(* Logix 5000 project; controller Safety vendor 1 type 14 code 148 rev 32.11; software revision 32.03; part 16 of 17 *)
(* tags used below, declared in another part *)
   A1_CoilCarSolPwrEn : BOOL;   // A1 UNW COIL CAR Solenoid Safe-Off Enable ( 1= Enable )
   A1_S20_ModFlt : ALIAS FOR Flt_Modules[0].0;   // A1 Point I/O Slot20 Module Fault (1 = Fault)
   A1_S21_ModFlt : ALIAS FOR Flt_Modules[0].1;   // A1 Point I/O Slot21 Module Fault (1 = Fault)
   C1_S12_ModFlt : ALIAS FOR Flt_Modules[0].2;   // C1 Point I/O Slot12 Module Fault (1 = Fault)
   CC : ALIAS FOR Diag_Tmp.0;   // Chris Como's Test Bit Always On Bit
   CHPLC_S1_ModFlt : ALIAS FOR Flt_Modules[0].3;   // CHPLC Point I/O Slot01 Module Fault (1 = Fault)
   CHPLC_S2_ModFlt : ALIAS FOR Flt_Modules[0].4;   // CHPLC Point I/O Slot02 Module Fault (1 = Fault)
   CHPLC_S3_ModFlt : ALIAS FOR Flt_Modules[0].5;   // CHPLC Point I/O Slot03 Module Fault (1 = Fault)
   CHPLC_S4_ModFlt : ALIAS FOR Flt_Modules[0].6;   // CHPLC Point I/O Slot04 Module Fault (1 = Fault)
   CHPLC_S5_ModFlt : ALIAS FOR Flt_Modules[0].7;   // CHPLC Point I/O Slot05 Module Fault (1 = Fault)
   CHPLC_S6_ModFlt : ALIAS FOR Flt_Modules[0].8;   // CHPLC Point I/O Slot06 Module Fault (1 = Fault)
   Citect_HB_Flt : BOOL;   // Citect Heartbeat Fault ( 1= Fault)
   Citect_HB_TOF : TIMER;   // Citect Heartbeat Timer Off
   Citect_HB_TON : TIMER;   // Citect Heartbeat Timer On
   D1_S12_ModFlt : ALIAS FOR Flt_Modules[0].9;   // D1 Point I/O Slot12 Module Fault (1 = Fault)
   DPD_No_EStops : BOOL;   // DPD No Estops ( 1= OK)
   DPD_S14_ModFlt : ALIAS FOR Flt_Modules[0].10;   // DPD Point I/O Slot14 Module Fault (1 = Fault)
   DPD_S15_ModFlt : ALIAS FOR Flt_Modules[0].11;   // DPD Point I/O Slot15 Module Fault (1 = Fault)
   Drives_Off : DINT;   // Line Drives Off
   E1_S10_ModFlt : ALIAS FOR Flt_Modules[0].12;   // E1 Point I/O Slot10 Module Fault (1 = Fault)
   EnBridle_DrvsOff : BOOL;   // Entry Bridle Drives OFF ( 1= OFF)
   ESTOP_x201PB040_Flt : ALIAS FOR Flt_Estops.0;   // OS1 Line EStop Pushbutton Fault ( 1= Fault)
   ESTOP_x211PB040_Flt : ALIAS FOR Flt_Estops.1;   // OS2 Line EStop Pushbutton Fault ( 1= Fault)
   ESTOP_x221PB040_Flt : ALIAS FOR Flt_Estops.2;   // OS3 Line EStop Pushbutton Fault ( 1= Fault)
   ESTOP_x231PB040_Flt : ALIAS FOR Flt_Estops.3;   // OS4N Line EStop Pushbutton Fault ( 1= Fault)
   ESTOP_x241PB040_Flt : ALIAS FOR Flt_Estops.4;   // OS4S Line EStop Pushbutton Fault ( 1= Fault)
   ESTOP_x251PB040_Flt : ALIAS FOR Flt_Estops.5;   // OS5 Line EStop Pushbutton Fault ( 1= Fault)
   ESTOP_x261PB040_Flt : ALIAS FOR Flt_Estops.6;   // OS6 Line EStop Pushbutton Fault ( 1= Fault)
   ESTOP_x271PB040_Flt : ALIAS FOR Flt_Estops.7;   // OS8 Line EStop Pushbutton Fault ( 1= Fault)
   ESTOP_x281PB040_Flt : ALIAS FOR Flt_Estops.8;   // OS9 Line EStop Pushbutton Fault ( 1= Fault)
   ESTOP_x291PB040_Flt : ALIAS FOR Flt_Estops.9;   // OS11 Line EStop Pushbutton Fault ( 1= Fault)
   ESTOP_x301PB040_Flt : ALIAS FOR Flt_Estops.10;   // OS13 Line EStop Pushbutton Fault ( 1= Fault)
   ESTOP_x311PB040_Flt : ALIAS FOR Flt_Estops.11;   // OS14 Line EStop Pushbutton Fault ( 1= Fault)
   ESTOP_x311PB130_Flt : ALIAS FOR Flt_Estops.17;   // OS14 Shear EStop Pushbutton Fault ( 1= Fault)
   ESTOP_x321PB040_Flt : ALIAS FOR Flt_Estops.12;   // OS15 Line EStop Pushbutton Fault ( 1= Fault)
   ESTOP_x331PB040_Flt : ALIAS FOR Flt_Estops.13;   // OS16 Line EStop Pushbutton Fault ( 1= Fault)
   ESTOP_x480PB470_Flt : ALIAS FOR Flt_Estops.14;   // DPD Line EStop Pushbutton Fault ( 1= Fault)
   ESTOP_x519LS470_Flt : ALIAS FOR Flt_Estops.18;   // G1 Line EStop Tripwire Limit Switch Fault ( 1= Fault)
   ESTOP_x533PB470_Flt : ALIAS FOR Flt_Estops.16;   // H1 Line EStop Pushbutton Fault ( 1= Fault)
   ExBridle_DrvsOff : BOOL;   // Exit Bridle Drives OFF ( 1= OFF)
   F1_S19_ModFlt : ALIAS FOR Flt_Modules[0].13;   // F1 Point I/O Slot19 Module Fault (1 = Fault)
   F1_S20_ModFlt : ALIAS FOR Flt_Modules[0].14;   // F1 Point I/O Slot20 Module Fault (1 = Fault)
   FromMachine : DINT[35];   // (FromMach)
   FromSafety : DINT[35];   // (From Safety)
   FromShearDie : DINT[35];   // (From Shear Die)
   FVR_y702MTR191_Flt : ALIAS FOR Flt_Starter.4;   // Rewind Pinch Roll Starter Fault ( 1= Fault)
   FVR_y708MTR080_Flt : ALIAS FOR Flt_Starter.1;   // Flattener Drive Motor Starter Fault ( 1= Fault)
   FVR_y708MTR250_Flt : ALIAS FOR Flt_Starter.0;   // Unwind Hold Down Roll Starter Fault ( 1= Fault)
   FVR_y753MTR190_Flt : ALIAS FOR Flt_Starter.2;   // Trimmer Pinch Roll Starter Fault ( 1= Fault)
   FVR_y761MTR081_Flt : ALIAS FOR Flt_Starter.3;   // Trimmer Scrap Conveyor Starter Fault ( 1= Fault)
   FVR_y778MTR080_Flt : ALIAS FOR Flt_Starter.5;   // Shear Die Crank Starter Fault ( 1= Fault)
   FVR_y802MTR080_Flt : ALIAS FOR Flt_Starter.6;   // Stacker Side Guide Lift Starter Fault ( 1= Fault)
   FVR_y802MTR230_Flt : ALIAS FOR Flt_Starter.8;   // Scrap Horizontal Conveyor Starter Fault ( 1= Fault)
   FVR_y802MTR231_Flt : ALIAS FOR Flt_Starter.7;   // Stacker Chain Conveyor Starter Fault ( 1= Fault)
   G1_No_EStops : BOOL;   // G1 No Estops ( 1= OK)
   G1_S11_ModFlt : ALIAS FOR Flt_Modules[0].15;   // G1 Point I/O Slot11 Module Fault (1 = Fault)
   G1_S12_ModFlt : ALIAS FOR Flt_Modules[0].16;   // G1 Point I/O Slot12 Module Fault (1 = Fault)
   H1_No_EStops : BOOL;   // H1 No Estops ( 1= OK)
   H1_S5_ModFlt : ALIAS FOR Flt_Modules[0].17;   // H1 Point I/O Slot05 Module Fault (1 = Fault)
   H1_S6_ModFlt : ALIAS FOR Flt_Modules[0].18;   // H1 Point I/O Slot06 Module Fault (1 = Fault)
   HB_Citect : BOOL;   // Heartbeat Citect Reflect
   Line_CTC_CoastStop : BOOL;   // Line Coast Stop ( 1= Coast Stop) (Condition Exists)
   Line_CTL_CoastStop : BOOL;   // Line Coast Stop ( 1= Coast Stop) (Condition Exists)
   Line_NoP2P_CommFlts : BOOL;   // Line No Peer to Peer Comm Faults ( 1= OK)
   Line_Total_CoastStop : BOOL;   // Line Coast Stop ( 1= Coast Stop) (Condition Exists)
   Line_TotalMode : BOOL;   // Line TOTAL Mode ( 1= Total Mode) (0 = Coil to Coil)
   LineSts : UDT_SysStatus;
   Machine_HB_Flt : BOOL;   // Machine Heartbeat Fault ( 1= Fault)
   Machine_HB_TOF : TIMER;   // Machine Heartbeat Timer Off
   Machine_HB_TON : TIMER;   // Machine Heartbeat Timer On
   MCC1_S1_ModFlt : ALIAS FOR Flt_Modules[2].0;   // MCC1 Point I/O Slot01 Module Fault (1 = Fault)
   MCC1_S6_ModFlt : ALIAS FOR Flt_Modules[2].1;   // MCC1 Point I/O Slot06 Module Fault (1 = Fault)
   MCC2_S1_ModFlt : ALIAS FOR Flt_Modules[2].2;   // MCC2 Point I/O Slot01 Module Fault (1 = Fault)
   MCC2_S2_ModFlt : ALIAS FOR Flt_Modules[2].3;   // MCC2 Point I/O Slot02 Module Fault (1 = Fault)
   MCC3_S1_ModFlt : ALIAS FOR Flt_Modules[2].4;   // MCC3 Point I/O Slot01 Module Fault (1 = Fault)
   MCC3_S3_ModFlt : ALIAS FOR Flt_Modules[2].5;   // MCC3 Point I/O Slot03 Module Fault (1 = Fault)
   MCC3_S4_ModFlt : ALIAS FOR Flt_Modules[2].6;   // MCC3 Point I/O Slot04 Module Fault (1 = Fault)
   MCC4_S1_ModFlt : ALIAS FOR Flt_Modules[2].7;   // MCC4 Point I/O Slot01 Module Fault (1 = Fault)
   MCC4_S3_ModFlt : ALIAS FOR Flt_Modules[2].8;   // MCC4 Point I/O Slot03 Module Fault (1 = Fault)
   MCC4_S4_ModFlt : ALIAS FOR Flt_Modules[2].9;   // MCC4 Point I/O Slot04 Module Fault (1 = Fault)
   MCC5_S1_ModFlt : ALIAS FOR Flt_Modules[2].10;   // MCC5 Point I/O Slot01 Module Fault (1 = Fault)
   MCC5_S3_ModFlt : ALIAS FOR Flt_Modules[2].11;   // MCC5 Point I/O Slot03 Module Fault (1 = Fault)
   MCC5_S4_ModFlt : ALIAS FOR Flt_Modules[2].12;   // MCC5 Point I/O Slot04 Module Fault (1 = Fault)
   MCC5_S5_ModFlt : ALIAS FOR Flt_Modules[2].13;   // MCC5 Point I/O Slot05 Module Fault (1 = Fault)
   OS11_No_EStops : BOOL;   // OS11 No Estops ( 1= OK)
   OS11_S1_ModFlt : ALIAS FOR Flt_Modules[1].11;   // OS11 Point I/O Slot01 Module Fault (1 = Fault)
   OS13_No_EStops : BOOL;   // OS13 No Estops ( 1= OK)
   OS13_S1_ModFlt : ALIAS FOR Flt_Modules[1].12;   // OS13 Point I/O Slot01 Module Fault (1 = Fault)
   OS14_No_EStops : BOOL;   // OS14 No Estops ( 1= OK)
   OS14_S1_ModFlt : ALIAS FOR Flt_Modules[1].13;   // OS14 Point I/O Slot01 Module Fault (1 = Fault)
   OS14_Shear_No_EStops : BOOL;   // OS14_Shear No Estops ( 1= OK)
   OS15_No_EStops : BOOL;   // OS15 No Estops ( 1= OK)
   OS15_S1_ModFlt : ALIAS FOR Flt_Modules[1].14;   // OS15 Point I/O Slot01 Module Fault (1 = Fault)
   OS16_No_EStops : BOOL;   // OS16 No Estops ( 1= OK)
   OS16_S1_ModFlt : ALIAS FOR Flt_Modules[1].15;   // OS16 Point I/O Slot01 Module Fault (1 = Fault)
   OS1_No_EStops : BOOL;   // OS1 No Estops ( 1= OK)
   OS1_S1_ModFlt : ALIAS FOR Flt_Modules[1].0;   // OS1 Point I/O Slot01 Module Fault (1 = Fault)
   OS2_No_EStops : BOOL;   // OS2 No Estops ( 1= OK)
   OS2_S1_ModFlt : ALIAS FOR Flt_Modules[1].1;   // OS2 Point I/O Slot01 Module Fault (1 = Fault)
   OS3_No_EStops : BOOL;   // OS3 No Estops ( 1= OK)
   OS3_S1_ModFlt : ALIAS FOR Flt_Modules[1].2;   // OS3 Point I/O Slot01 Module Fault (1 = Fault)
   OS4_No_EStops : BOOL;   // OS4 No Estops ( 1= OK)
   OS4N_S1_ModFlt : ALIAS FOR Flt_Modules[1].3;   // OS4N Point I/O Slot01 Module Fault (1 = Fault)
   OS4N_S5_ModFlt : ALIAS FOR Flt_Modules[1].4;   // OS4N Point I/O Slot05 Module Fault (1 = Fault)
   OS4S_S1_ModFlt : ALIAS FOR Flt_Modules[1].5;   // OS4S Point I/O Slot01 Module Fault (1 = Fault)
   OS4S_S5_ModFlt : ALIAS FOR Flt_Modules[1].6;   // OS4S Point I/O Slot05 Module Fault (1 = Fault)
   OS5_No_EStops : BOOL;   // OS5 No Estops ( 1= OK)
   OS5_S1_ModFlt : ALIAS FOR Flt_Modules[1].7;   // OS5 Point I/O Slot01 Module Fault (1 = Fault)
   OS6_No_EStops : BOOL;   // OS6 No Estops ( 1= OK)
   OS6_S1_ModFlt : ALIAS FOR Flt_Modules[1].8;   // OS6 Point I/O Slot01 Module Fault (1 = Fault)
   OS8_No_EStops : BOOL;   // OS8 No Estops ( 1= OK)
   OS8_S1_ModFlt : ALIAS FOR Flt_Modules[1].9;   // OS8 Point I/O Slot01 Module Fault (1 = Fault)
   OS9_No_EStops : BOOL;   // OS9 No Estops ( 1= OK)
   OS9_S1_ModFlt : ALIAS FOR Flt_Modules[1].10;   // OS9 Point I/O Slot01 Module Fault (1 = Fault)
   PrCon_DrvsOff : BOOL;   // Product Conveyors (1-3) Drives OFF ( 1= OFF)
   PW_DrvsOff : BOOL;   // Paper Winder Drives OFF ( 1= OFF)
   Rew_DrvsOff : BOOL;   // Rewind Drives OFF ( 1= OFF)
   SafeOff_y172CR460_Flt : ALIAS FOR Flt_SafeOff[0].0;   // Shear Die Main Contactor Relay Fault ( 1= Fault)
   SafeOff_y172CR510_Flt : ALIAS FOR Flt_SafeOff[0].1;   // Shear Die Drive Enable Relay Fault ( 1= Fault)
   SafeOff_y613CR460_Flt : ALIAS FOR Flt_SafeOff[0].2;   // Unwind Op Side Main Contactor Relay Fault ( 1= Fault)
   SafeOff_y613CR510_Flt : ALIAS FOR Flt_SafeOff[0].3;   // Unwind Op Side Drive Enable Relay Fault ( 1= Fault)
   SafeOff_y613CR550_Flt : ALIAS FOR Flt_SafeOff[0].4;   // Unwind Drive Side Main Contactor Relay Fault ( 1= Fault)
   SafeOff_y613CR590_Flt : ALIAS FOR Flt_SafeOff[0].5;   // Unwind Drive Side Drive Enable Relay Fault ( 1= Fault)
   SafeOff_y613CR630_Flt : ALIAS FOR Flt_SafeOff[0].6;   // #1 Entry Bridle Roll 2 Main Contactor Relay Fault ( 1= Fault)
   SafeOff_y613CR670_Flt : ALIAS FOR Flt_SafeOff[0].7;   // #1 Entry Bridle Roll 2 Drive Enable Relay Fault ( 1= Fault)
   SafeOff_y613CR710_Flt : ALIAS FOR Flt_SafeOff[0].8;   // #2 Entry Bridle Roll 3 Main Contactor Relay Fault ( 1= Fault)
   SafeOff_y613CR750_Flt : ALIAS FOR Flt_SafeOff[0].9;   // #2 Entry Bridle Roll 3 Drive Enable Relay Fault ( 1= Fault)
   SafeOff_y614CR040_Flt : ALIAS FOR Flt_SafeOff[0].10;   // #1 Exit Bridle Roll 6 Main Contactor Relay Fault ( 1= Fault)
   SafeOff_y614CR090_Flt : ALIAS FOR Flt_SafeOff[0].11;   // #1 Exit Bridle Roll 6 Drive Enable Relay Fault ( 1= Fault)
   SafeOff_y614CR130_Flt : ALIAS FOR Flt_SafeOff[0].12;   // #2 Exit Bridle Roll 7 Main Contactor Relay Fault ( 1= Fault)
   SafeOff_y614CR170_Flt : ALIAS FOR Flt_SafeOff[0].13;   // #2 Exit Bridle Roll 7 Drive Enable Relay Fault ( 1= Fault)
   SafeOff_y614CR210_Flt : ALIAS FOR Flt_SafeOff[0].14;   // Rewind Main Contactor Relay Fault ( 1= Fault)
   SafeOff_y614CR250_Flt : ALIAS FOR Flt_SafeOff[0].15;   // Rewind Drive Enable Relay Fault ( 1= Fault)
   Safety_HB_TOF : TIMER;   // Safety Heartbeat Pulse Time Off
   Safety_HB_TON : TIMER;   // Safety Heartbeat Pulse Time On
   SC_DrvsOff : BOOL;   // Scrap Chop Conveyor Drives OFF ( 1= OFF)
   ScInCon_DrvsOff : BOOL;   // Scrap Incline Conveyor Drives OFF ( 1= OFF)
   SDPLC_S1_ModFlt : ALIAS FOR Flt_Modules[0].19;   // SDPLC Point I/O Slot01 Module Fault (1 = Fault)
   SDPLC_S2_ModFlt : ALIAS FOR Flt_Modules[0].20;   // SDPLC Point I/O Slot02 Module Fault (1 = Fault)
   Sfty_InstrFlts0_CTC : BOOL;   // Coil To Coil Estop Safety Instructions OK ( 1= No Faults)
   Sfty_InstrFlts0_CTL : BOOL;   // Cut To Length Estop Safety Instructions OK ( 1= No Faults)
   Sfty_InstrFlts0_Total : BOOL;   // Total Mode Estop Safety Instructions OK ( 1= No Faults)
   Sfty_InstrFlts1_CTC : BOOL;   // Coil To Coil Safe-Off Safety Instructions OK ( 1= No Faults)
   Sfty_InstrFlts1_CTL : BOOL;   // Cut To Length Safe-Off Safety Instructions OK ( 1= No Faults)
   Sfty_InstrFlts1_Total : BOOL;   // Total Mode Safe-Off Safety Instructions OK ( 1= No Faults)
   Sfty_InstrFlts2_CTC : BOOL;   // Coil To Coil FVR/FVNR Starters Safety Instructions OK ( 1= No Faults)
   Sfty_InstrFlts2_CTL : BOOL;   // Cut To Length FVR/FVNR Starters Safety Instructions OK ( 1= No Faults)
   Sfty_InstrFlts2_Total : BOOL;   // Total Mode FVR/FVNR Starters Safety Instructions OK ( 1= No Faults)
   Sfty_ModFlts0_CTC : BOOL;   // Coil To Coil General I/O Safety Module Faults ( 1= OK)
   Sfty_ModFlts0_CTL : BOOL;   // Cut To Length General I/O Safety Module Faults ( 1= OK)
   Sfty_ModFlts0_Total : BOOL;   // Total Mode General I/O Safety Module Faults ( 1= OK)
   Sfty_ModFlts1_CTC : BOOL;   // Coil To Coil Operator Station Safety Module Faults ( 1= OK)
   Sfty_ModFlts1_CTL : BOOL;   // Cut To Length Operator Station Safety Module Faults ( 1= OK)
   Sfty_ModFlts1_Total : BOOL;   // Total Mode Operator Station Safety Module Faults ( 1= OK)
   Sfty_ModFlts2_CTC : BOOL;   // Coil To Coil MCC Safety Module Faults ( 1= OK)
   Sfty_ModFlts2_CTL : BOOL;   // Cut To Lenght MCC Safety Module Faults ( 1= OK)
   Sfty_ModFlts2_Total : BOOL;   // Total Mode MCC Safety Module Faults ( 1= OK)
   SftyMap_Citect : DINT[5];   // SAFETY MAPPED From Citect System
   SftyMap_Mach : DINT[5];   // SAFETY MAPPED From Machine Processor
   SftyMap_ShDie : DINT[5];   // SAFETY MAPPED From Shear Die Processor
   SGWA_DrvsOff : BOOL;   // Side Guide Width Adjust Drives OFF ( 1= OFF)
   Shear_CoastStop : BOOL;   // Shear Coast Stop ( 1= Coast Stop) (Condition Exists)
   Shear_HB_Flt : BOOL;   // Shear Heartbeat Fault ( 1= Fault)
   Shear_HB_TOF : TIMER;   // Shear Heartbeat Pulse Time Off
   Shear_HB_TON : TIMER;   // Shear Heartbeat Pulse Time On
   ShearSts : UDT_ShearStatus;
   SkBkSt_DrvsOff : BOOL;   // Stacker Backstop Drives OFF ( 1= OFF)
   SkBlwr_DrvsOff : BOOL;   // Stacker Blower Drives OFF ( 1= OFF)
   Sr_DrvsOff : BOOL;   // Shear Pinch Roll/ Metering Back Up Drives OFF ( 1= OFF)
   SrCon_DrvsOff : BOOL;   // Shear Conveyor Drives OFF ( 1= OFF)
   SrDie_DrvsOff : BOOL;   // Shear Die Drives OFF ( 1= OFF)
   StPR_DrvsOff : BOOL;   // Sheeter Pinch Roll Drives OFF ( 1= OFF)
   TK_DrvsOff : BOOL;   // Trimmer Knives/ Width Adjust Drives OFF ( 1= OFF)
   ToCitect : DINT[64];   // (To Citect)
   UnPR_DrvsOff : BOOL;   // Unwind Pinch Roll Drives OFF ( 1= OFF)
   UNW_DrvsOff : BOOL;   // Unwind Drives OFF ( 1= OFF)
   VS2_S10_ModFlt : ALIAS FOR Flt_Modules[0].21;   // VS2 Point I/O Slot10 Module Fault (1 = Fault)
   WTPR_DrvsOff : BOOL;   // Wash Tank Pinch Rolls (1-4) Drives OFF ( 1= OFF)
(* System, continued *)

ROUTINE A04_SftyHeartbeat   (* ladder *)
// Heartbeat Logic
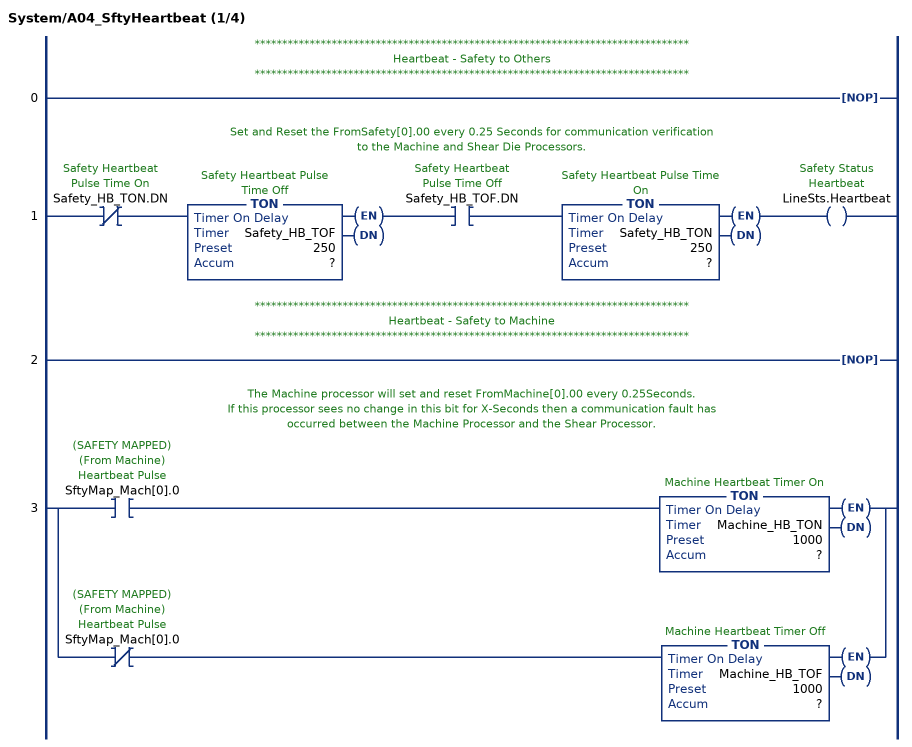
   // *******************************************************************************
   // Heartbeat - Safety to Others
   // *******************************************************************************
   0: NOP();
   // Set and Reset the FromSafety[0].00 every 0.25 Seconds for communication verification
   // to the Machine and Shear Die Processors.
   1: XIO(Safety_HB_TON.DN)TON(Safety_HB_TOF,?,?)XIC(Safety_HB_TOF.DN)TON(Safety_HB_TON,?,?)OTE(LineSts.Heartbeat);
   // *******************************************************************************
   // Heartbeat - Safety to Machine
   // *******************************************************************************
   2: NOP();
   // The Machine processor will set and reset FromMachine[0].00 every 0.25Seconds.
   // If this processor sees no change in this bit for X-Seconds then a communication fault has
   // occurred between the Machine Processor and the Shear Processor.
   3: [XIC(SftyMap_Mach[0].0) TON(Machine_HB_TON,?,?) ,XIO(SftyMap_Mach[0].0) TON(Machine_HB_TOF,?,?) ];
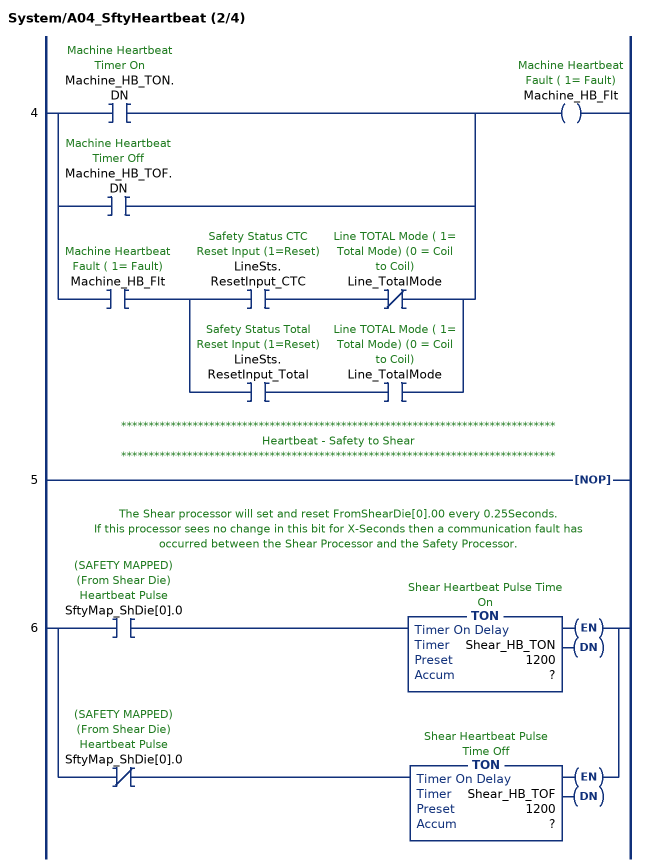
   4: [XIC(Machine_HB_TON.DN) ,XIC(Machine_HB_TOF.DN) ,XIC(Machine_HB_Flt) [XIC(LineSts.ResetInput_CTC) XIO(Line_TotalMode) ,XIC(LineSts.ResetInput_Total) XIC(Line_TotalMode) ] ]OTE(Machine_HB_Flt);
   // *******************************************************************************
   // Heartbeat - Safety to Shear
   // *******************************************************************************
   5: NOP();
   // The Shear processor will set and reset FromShearDie[0].00 every 0.25Seconds.
   // If this processor sees no change in this bit for X-Seconds then a communication fault has
   // occurred between the Shear Processor and the Safety Processor.
   6: [XIC(SftyMap_ShDie[0].0) TON(Shear_HB_TON,?,?) ,XIO(SftyMap_ShDie[0].0) TON(Shear_HB_TOF,?,?) ];
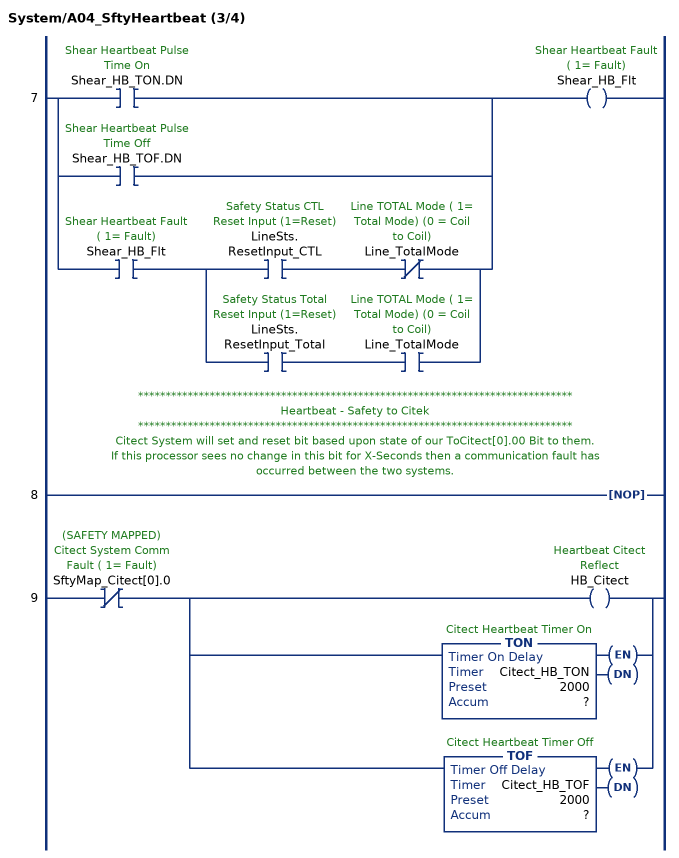
   7: [XIC(Shear_HB_TON.DN) ,XIC(Shear_HB_TOF.DN) ,XIC(Shear_HB_Flt) [XIC(LineSts.ResetInput_CTL) XIO(Line_TotalMode) ,XIC(LineSts.ResetInput_Total) XIC(Line_TotalMode) ] ]OTE(Shear_HB_Flt);
   // *******************************************************************************
   // Heartbeat - Safety to Citek
   // *******************************************************************************
   // Citect System will set and reset bit based upon state of our ToCitect[0].00 Bit to them.
   // If this processor sees no change in this bit for X-Seconds then a communication fault has
   // occurred between the two systems.
   8: NOP();
   9: XIO(SftyMap_Citect[0].0)[OTE(HB_Citect) ,TON(Citect_HB_TON,?,?) ,TOF(Citect_HB_TOF,?,?) ];
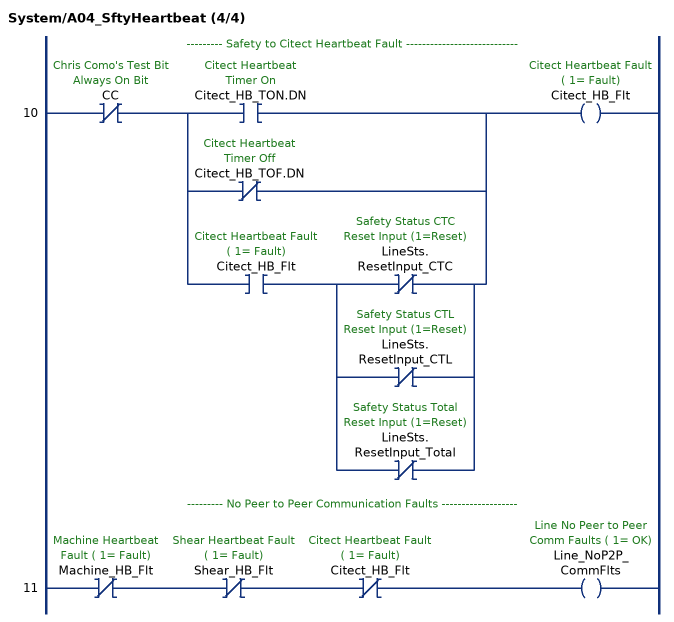
   // --------- Safety to Citect Heartbeat Fault ----------------------------
   10: XIO(CC)[XIC(Citect_HB_TON.DN) ,XIO(Citect_HB_TOF.DN) ,XIC(Citect_HB_Flt) [XIO(LineSts.ResetInput_CTC) ,XIO(LineSts.ResetInput_CTL) ,XIO(LineSts.ResetInput_Total) ] ]OTE(Citect_HB_Flt);
   // --------- No Peer to Peer Communication Faults -------------------
   11: XIO(Machine_HB_Flt)XIO(Shear_HB_Flt)XIO(Citect_HB_Flt)OTE(Line_NoP2P_CommFlts);
END_ROUTINE

ROUTINE B00_Line_Logic   (* ladder *)
// Line System
// Safety Logic
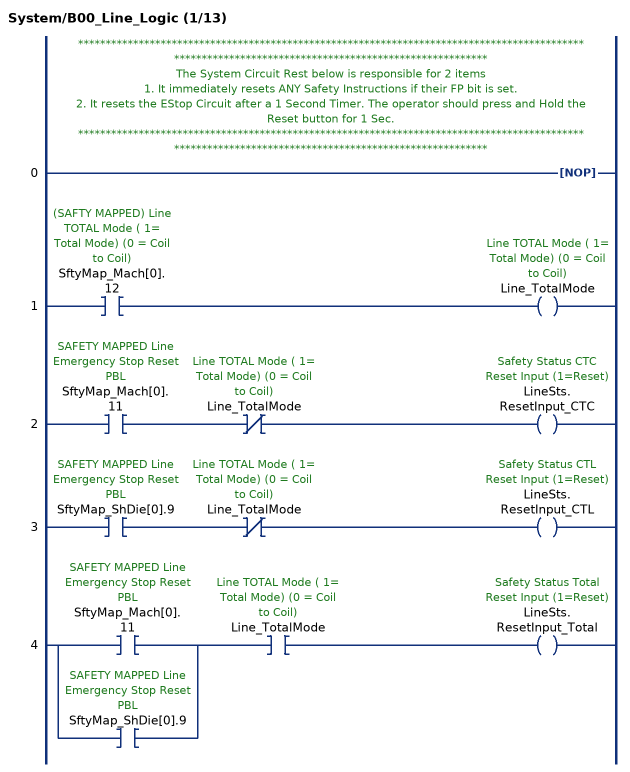
   // *****************************************************************************************************************************************************
   // The System Circuit Rest below is responsible for 2 items
   // 1. It immediately resets ANY Safety Instructions if their FP bit is set.
   // 2. It resets the EStop Circuit after a 1 Second Timer. The operator should press and Hold the Reset button for 1 Sec.
   // *****************************************************************************************************************************************************
   0: NOP();
   1: XIC(SftyMap_Mach[0].12)OTE(Line_TotalMode);
   2: XIC(SftyMap_Mach[0].11)XIO(Line_TotalMode)OTE(LineSts.ResetInput_CTC);
   3: XIC(SftyMap_ShDie[0].9)XIO(Line_TotalMode)OTE(LineSts.ResetInput_CTL);
   4: [XIC(SftyMap_Mach[0].11) ,XIC(SftyMap_ShDie[0].9) ]XIC(Line_TotalMode)OTE(LineSts.ResetInput_Total);
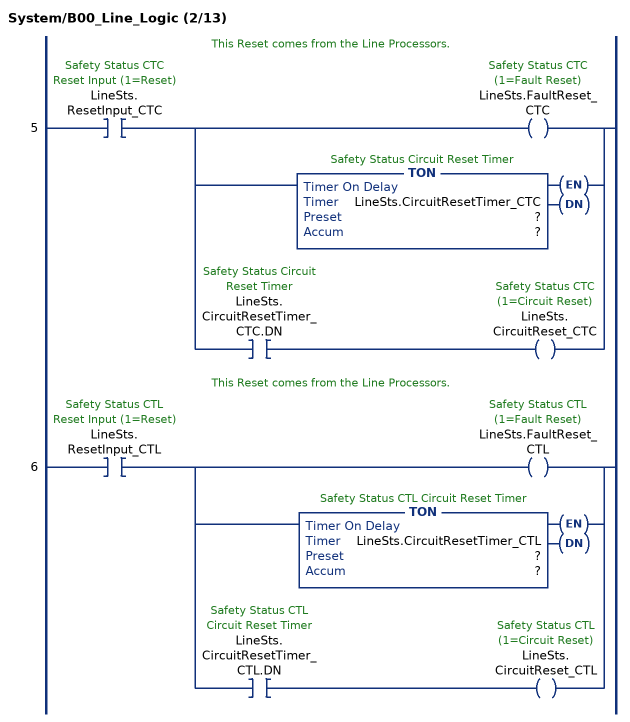
   // This Reset comes from the Line Processors.
   5: XIC(LineSts.ResetInput_CTC)[OTE(LineSts.FaultReset_CTC) ,TON(LineSts.CircuitResetTimer_CTC,?,?) ,XIC(LineSts.CircuitResetTimer_CTC.DN) OTE(LineSts.CircuitReset_CTC) ];
   // This Reset comes from the Line Processors.
   6: XIC(LineSts.ResetInput_CTL)[OTE(LineSts.FaultReset_CTL) ,TON(LineSts.CircuitResetTimer_CTL,?,?) ,XIC(LineSts.CircuitResetTimer_CTL.DN) OTE(LineSts.CircuitReset_CTL) ];
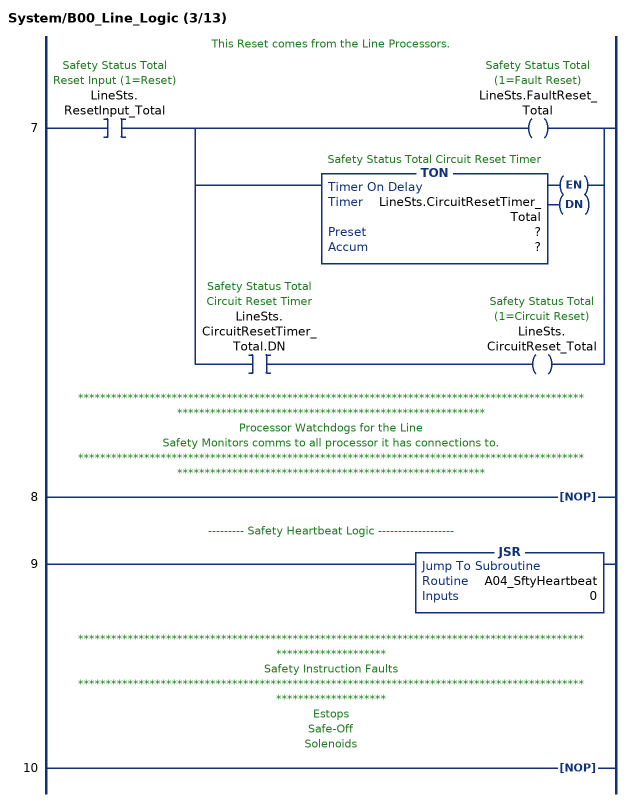
   // This Reset comes from the Line Processors.
   7: XIC(LineSts.ResetInput_Total)[OTE(LineSts.FaultReset_Total) ,TON(LineSts.CircuitResetTimer_Total,?,?) ,XIC(LineSts.CircuitResetTimer_Total.DN) OTE(LineSts.CircuitReset_Total) ];
   // ****************************************************************************************************************************************************
   // Processor Watchdogs for the Line
   // Safety Monitors comms to all processor it has connections to.
   // ****************************************************************************************************************************************************
   8: NOP();
   // --------- Safety Heartbeat Logic -------------------
   9: JSR(A04_SftyHeartbeat,0);
   // ****************************************************************************************************************
   // Safety Instruction Faults
   // ****************************************************************************************************************
   // Estops
   // Safe-Off
   // Solenoids
   10: NOP();
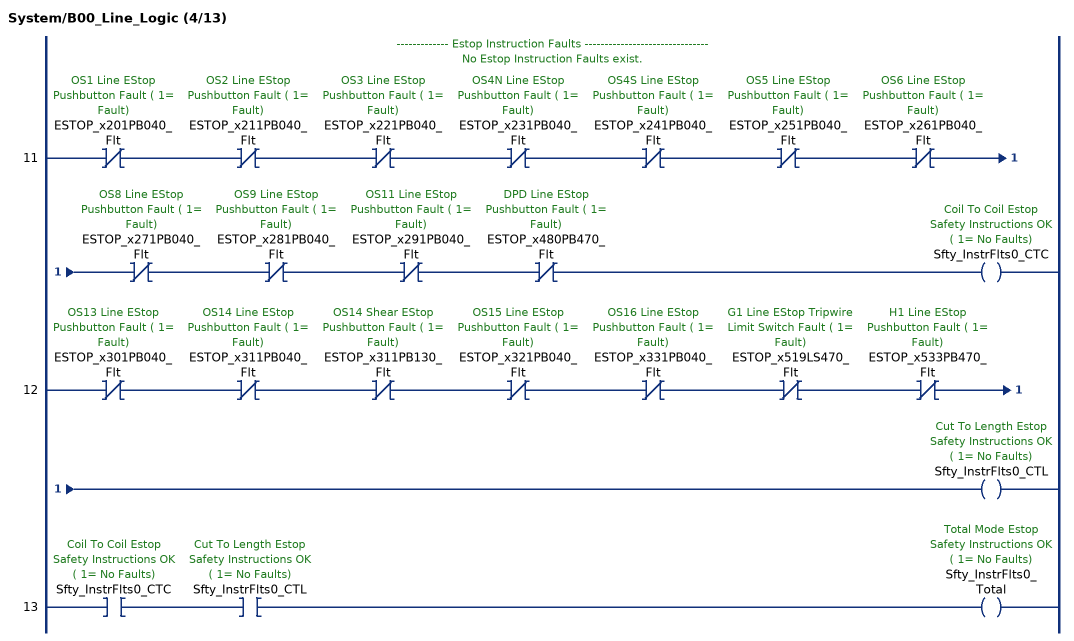
   // ------------- Estop Instruction Faults -------------------------------
   // No Estop Instruction Faults exist.
   11: XIO(ESTOP_x201PB040_Flt)XIO(ESTOP_x211PB040_Flt)XIO(ESTOP_x221PB040_Flt)XIO(ESTOP_x231PB040_Flt)XIO(ESTOP_x241PB040_Flt)XIO(ESTOP_x251PB040_Flt)XIO(ESTOP_x261PB040_Flt)XIO(ESTOP_x271PB040_Flt)XIO(ESTOP_x281PB040_Flt)XIO(ESTOP_x291PB040_Flt)XIO(ESTOP_x480PB470_Flt)OTE(Sfty_InstrFlts0_CTC);
   12: XIO(ESTOP_x301PB040_Flt)XIO(ESTOP_x311PB040_Flt)XIO(ESTOP_x311PB130_Flt)XIO(ESTOP_x321PB040_Flt)XIO(ESTOP_x331PB040_Flt)XIO(ESTOP_x519LS470_Flt)XIO(ESTOP_x533PB470_Flt)OTE(Sfty_InstrFlts0_CTL);
   13: XIC(Sfty_InstrFlts0_CTC)XIC(Sfty_InstrFlts0_CTL)OTE(Sfty_InstrFlts0_Total);
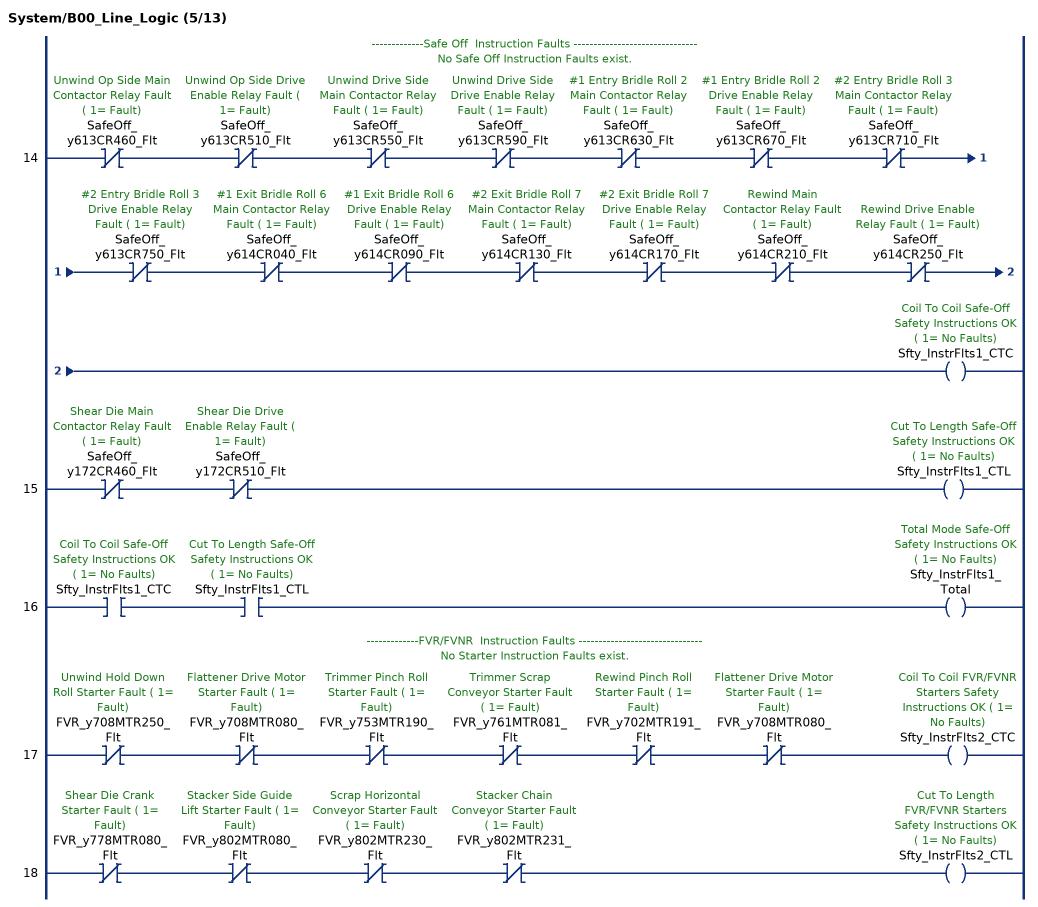
   // -------------Safe Off  Instruction Faults -------------------------------
   // No Safe Off Instruction Faults exist.
   14: XIO(SafeOff_y613CR460_Flt)XIO(SafeOff_y613CR510_Flt)XIO(SafeOff_y613CR550_Flt)XIO(SafeOff_y613CR590_Flt)XIO(SafeOff_y613CR630_Flt)XIO(SafeOff_y613CR670_Flt)XIO(SafeOff_y613CR710_Flt)XIO(SafeOff_y613CR750_Flt)XIO(SafeOff_y614CR040_Flt)XIO(SafeOff_y614CR090_Flt)XIO(SafeOff_y614CR130_Flt)XIO(SafeOff_y614CR170_Flt)XIO(SafeOff_y614CR210_Flt)XIO(SafeOff_y614CR250_Flt)OTE(Sfty_InstrFlts1_CTC);
   15: XIO(SafeOff_y172CR460_Flt)XIO(SafeOff_y172CR510_Flt)OTE(Sfty_InstrFlts1_CTL);
   16: XIC(Sfty_InstrFlts1_CTC)XIC(Sfty_InstrFlts1_CTL)OTE(Sfty_InstrFlts1_Total);
   // -------------FVR/FVNR  Instruction Faults -------------------------------
   // No Starter Instruction Faults exist.
   17: XIO(FVR_y708MTR250_Flt)XIO(FVR_y708MTR080_Flt)XIO(FVR_y753MTR190_Flt)XIO(FVR_y761MTR081_Flt)XIO(FVR_y702MTR191_Flt)XIO(FVR_y708MTR080_Flt)OTE(Sfty_InstrFlts2_CTC);
   18: XIO(FVR_y778MTR080_Flt)XIO(FVR_y802MTR080_Flt)XIO(FVR_y802MTR230_Flt)XIO(FVR_y802MTR231_Flt)OTE(Sfty_InstrFlts2_CTL);
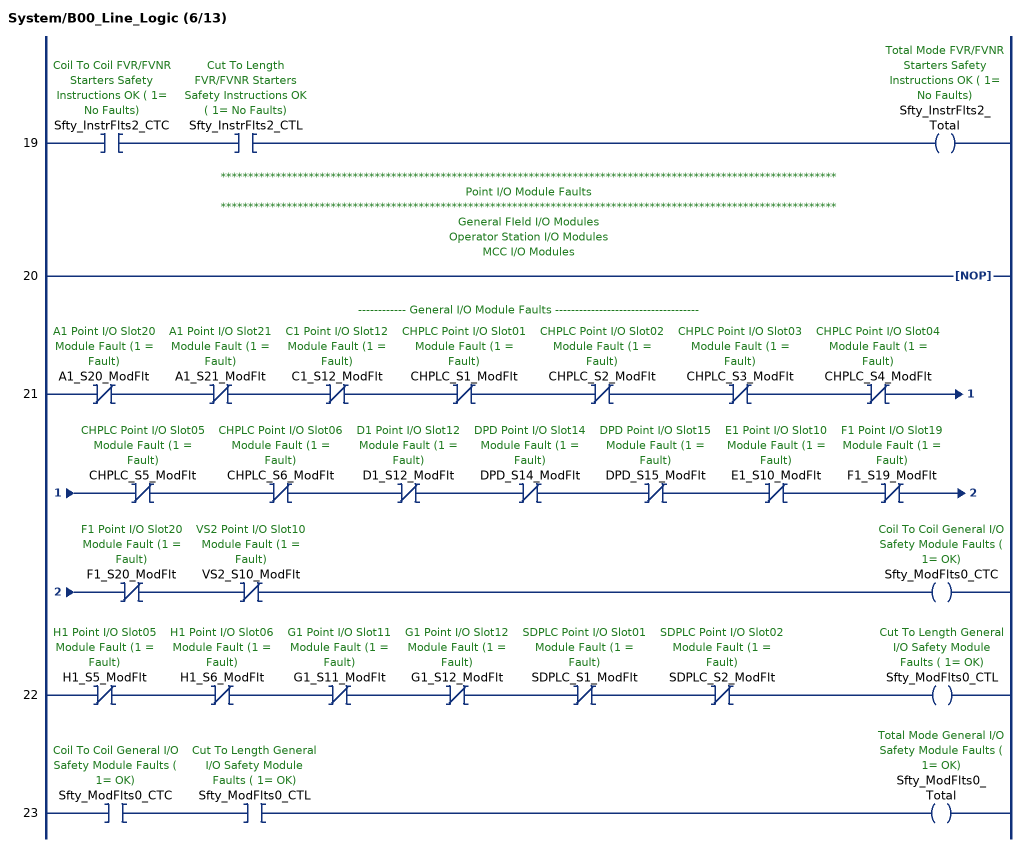
   19: XIC(Sfty_InstrFlts2_CTC)XIC(Sfty_InstrFlts2_CTL)OTE(Sfty_InstrFlts2_Total);
   // ****************************************************************************************************************
   // Point I/O Module Faults
   // ****************************************************************************************************************
   // General FIeld I/O Modules
   // Operator Station I/O Modules
   // MCC I/O Modules
   20: NOP();
   // ------------ General I/O Module Faults ------------------------------------
   21: XIO(A1_S20_ModFlt)XIO(A1_S21_ModFlt)XIO(C1_S12_ModFlt)XIO(CHPLC_S1_ModFlt)XIO(CHPLC_S2_ModFlt)XIO(CHPLC_S3_ModFlt)XIO(CHPLC_S4_ModFlt)XIO(CHPLC_S5_ModFlt)XIO(CHPLC_S6_ModFlt)XIO(D1_S12_ModFlt)XIO(DPD_S14_ModFlt)XIO(DPD_S15_ModFlt)XIO(E1_S10_ModFlt)XIO(F1_S19_ModFlt)XIO(F1_S20_ModFlt)XIO(VS2_S10_ModFlt)OTE(Sfty_ModFlts0_CTC);
   22: XIO(H1_S5_ModFlt)XIO(H1_S6_ModFlt)XIO(G1_S11_ModFlt)XIO(G1_S12_ModFlt)XIO(SDPLC_S1_ModFlt)XIO(SDPLC_S2_ModFlt)OTE(Sfty_ModFlts0_CTL);
   23: XIC(Sfty_ModFlts0_CTC)XIC(Sfty_ModFlts0_CTL)OTE(Sfty_ModFlts0_Total);
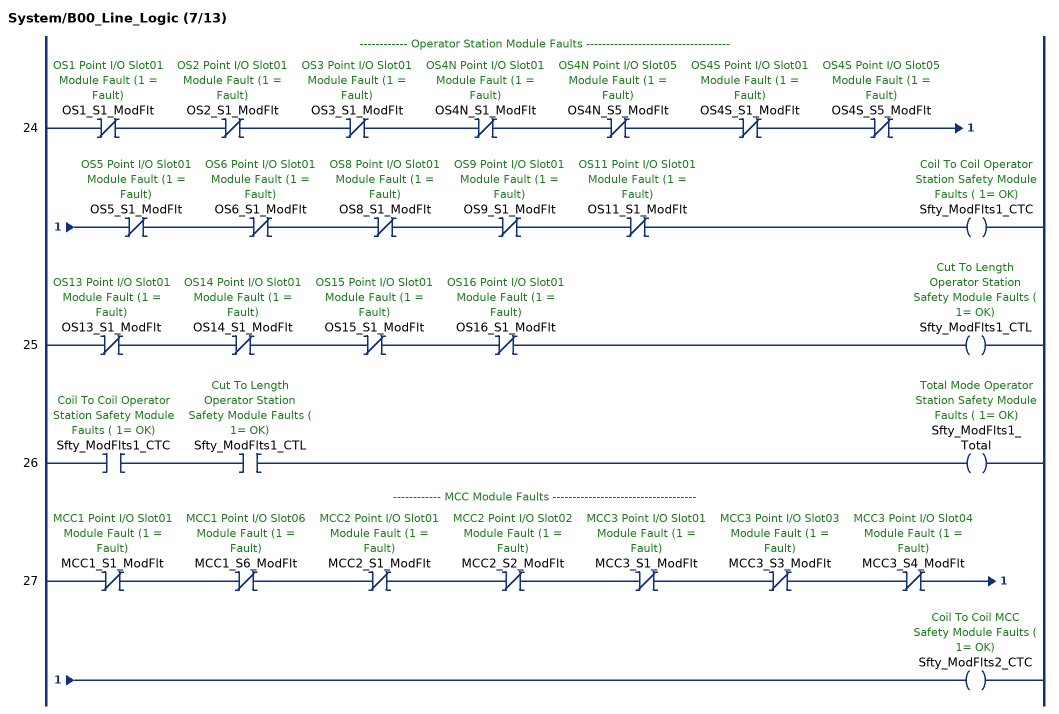
   // ------------ Operator Station Module Faults ------------------------------------
   24: XIO(OS1_S1_ModFlt)XIO(OS2_S1_ModFlt)XIO(OS3_S1_ModFlt)XIO(OS4N_S1_ModFlt)XIO(OS4N_S5_ModFlt)XIO(OS4S_S1_ModFlt)XIO(OS4S_S5_ModFlt)XIO(OS5_S1_ModFlt)XIO(OS6_S1_ModFlt)XIO(OS8_S1_ModFlt)XIO(OS9_S1_ModFlt)XIO(OS11_S1_ModFlt)OTE(Sfty_ModFlts1_CTC);
   25: XIO(OS13_S1_ModFlt)XIO(OS14_S1_ModFlt)XIO(OS15_S1_ModFlt)XIO(OS16_S1_ModFlt)OTE(Sfty_ModFlts1_CTL);
   26: XIC(Sfty_ModFlts1_CTC)XIC(Sfty_ModFlts1_CTL)OTE(Sfty_ModFlts1_Total);
   // ------------ MCC Module Faults ------------------------------------
   27: XIO(MCC1_S1_ModFlt)XIO(MCC1_S6_ModFlt)XIO(MCC2_S1_ModFlt)XIO(MCC2_S2_ModFlt)XIO(MCC3_S1_ModFlt)XIO(MCC3_S3_ModFlt)XIO(MCC3_S4_ModFlt)OTE(Sfty_ModFlts2_CTC);
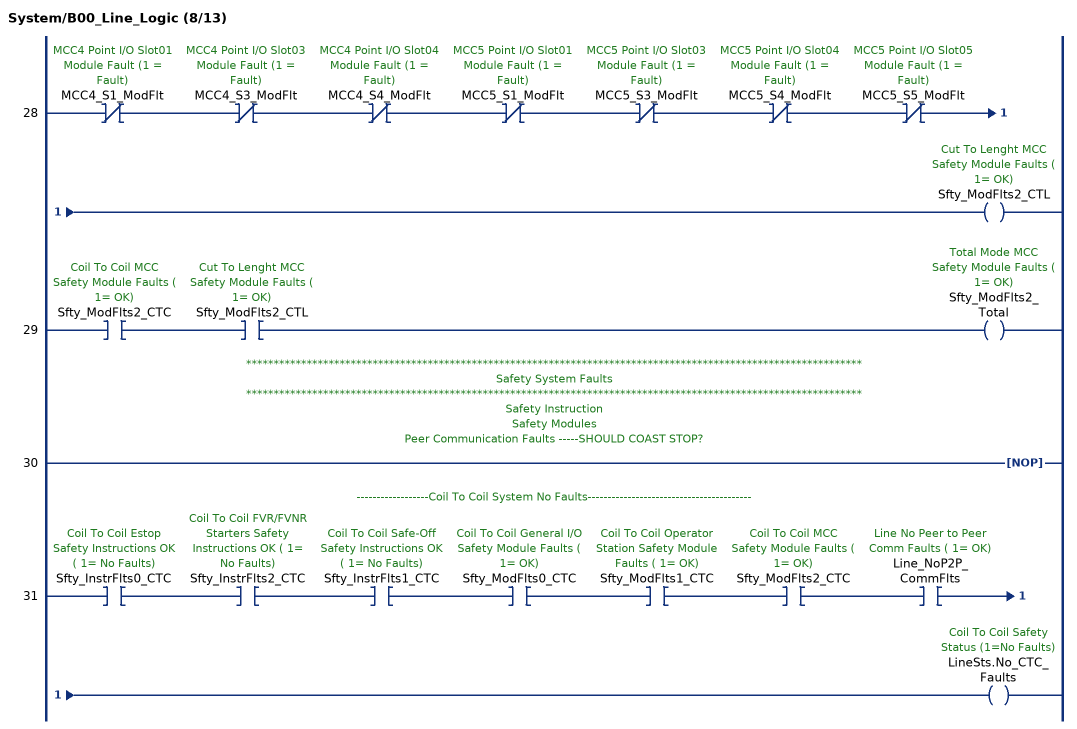
   28: XIO(MCC4_S1_ModFlt)XIO(MCC4_S3_ModFlt)XIO(MCC4_S4_ModFlt)XIO(MCC5_S1_ModFlt)XIO(MCC5_S3_ModFlt)XIO(MCC5_S4_ModFlt)XIO(MCC5_S5_ModFlt)OTE(Sfty_ModFlts2_CTL);
   29: XIC(Sfty_ModFlts2_CTC)XIC(Sfty_ModFlts2_CTL)OTE(Sfty_ModFlts2_Total);
   // ****************************************************************************************************************
   // Safety System Faults
   // ****************************************************************************************************************
   // Safety Instruction
   // Safety Modules
   // Peer Communication Faults -----SHOULD COAST STOP?
   30: NOP();
   // ------------------Coil To Coil System No Faults-----------------------------------------
   31: XIC(Sfty_InstrFlts0_CTC)XIC(Sfty_InstrFlts2_CTC)XIC(Sfty_InstrFlts1_CTC)XIC(Sfty_ModFlts0_CTC)XIC(Sfty_ModFlts1_CTC)XIC(Sfty_ModFlts2_CTC)XIC(Line_NoP2P_CommFlts)OTE(LineSts.No_CTC_Faults);
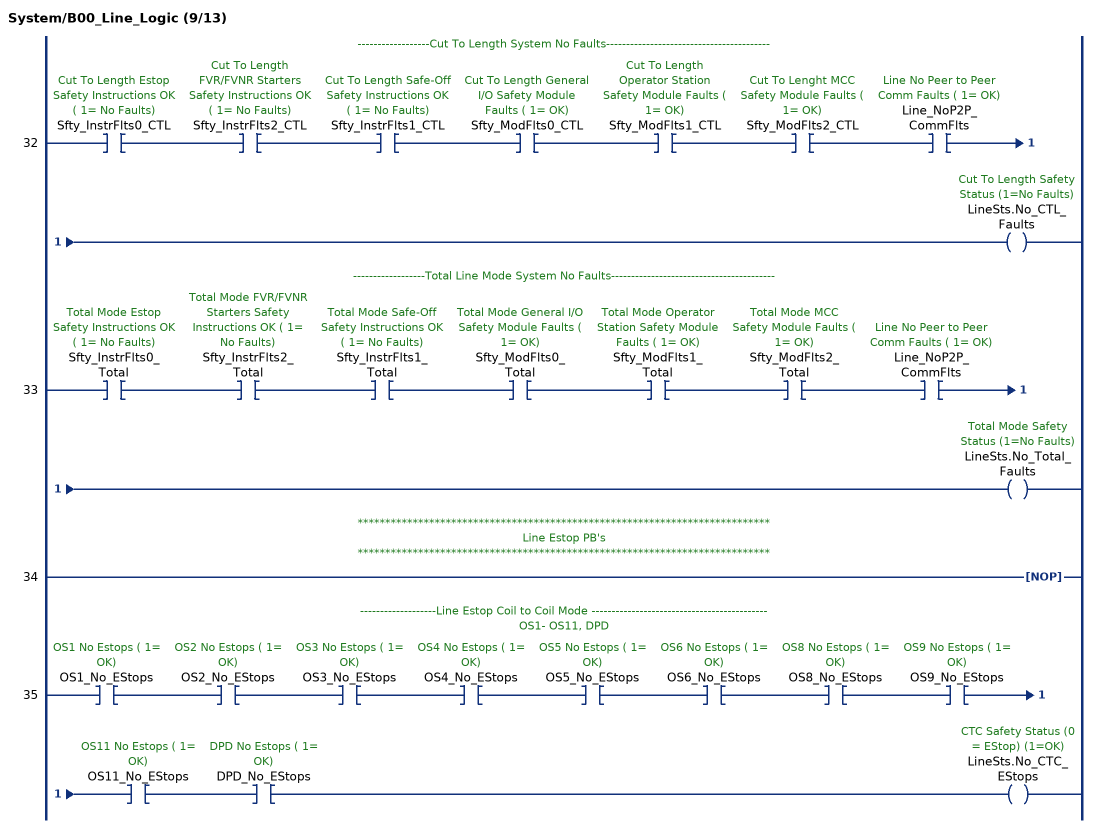
   // ------------------Cut To Length System No Faults-----------------------------------------
   32: XIC(Sfty_InstrFlts0_CTL)XIC(Sfty_InstrFlts2_CTL)XIC(Sfty_InstrFlts1_CTL)XIC(Sfty_ModFlts0_CTL)XIC(Sfty_ModFlts1_CTL)XIC(Sfty_ModFlts2_CTL)XIC(Line_NoP2P_CommFlts)OTE(LineSts.No_CTL_Faults);
   // ------------------Total Line Mode System No Faults-----------------------------------------
   33: XIC(Sfty_InstrFlts0_Total)XIC(Sfty_InstrFlts2_Total)XIC(Sfty_InstrFlts1_Total)XIC(Sfty_ModFlts0_Total)XIC(Sfty_ModFlts1_Total)XIC(Sfty_ModFlts2_Total)XIC(Line_NoP2P_CommFlts)OTE(LineSts.No_Total_Faults);
   // ***************************************************************************
   // Line Estop PB's
   // ***************************************************************************
   34: NOP();
   // -------------------Line Estop Coil to Coil Mode --------------------------------------------
   // OS1- OS11, DPD
   35: XIC(OS1_No_EStops)XIC(OS2_No_EStops)XIC(OS3_No_EStops)XIC(OS4_No_EStops)XIC(OS5_No_EStops)XIC(OS6_No_EStops)XIC(OS8_No_EStops)XIC(OS9_No_EStops)XIC(OS11_No_EStops)XIC(DPD_No_EStops)OTE(LineSts.No_CTC_EStops);
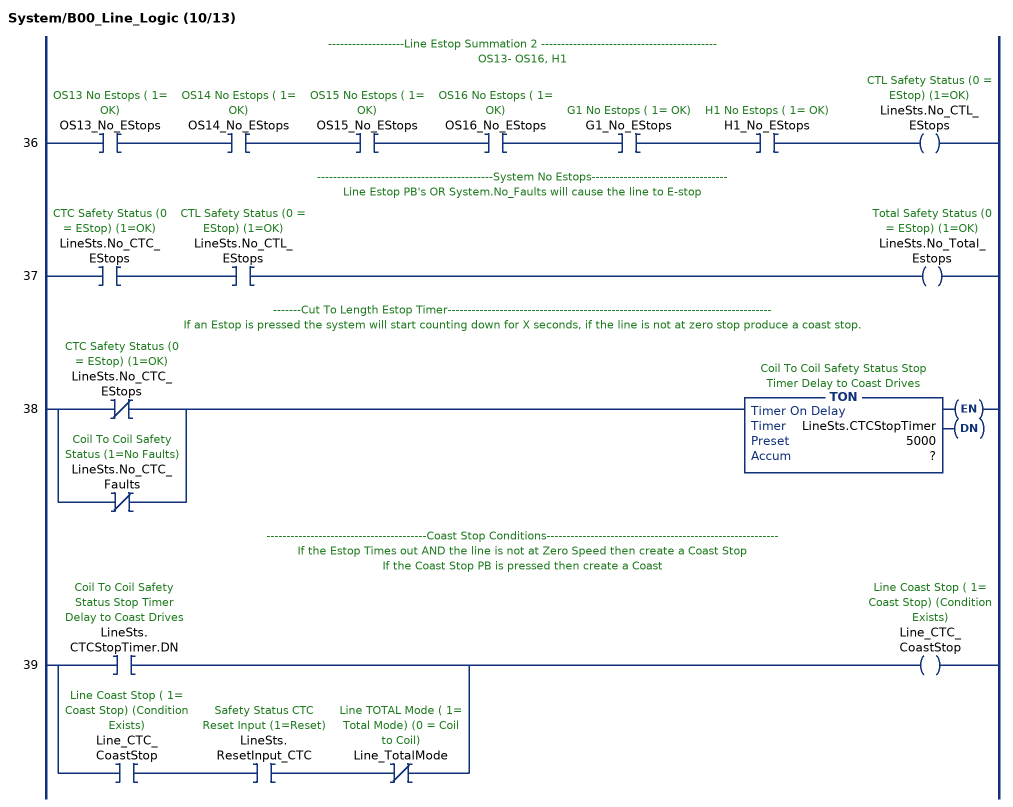
   // -------------------Line Estop Summation 2 --------------------------------------------
   // OS13- OS16, H1
   36: XIC(OS13_No_EStops)XIC(OS14_No_EStops)XIC(OS15_No_EStops)XIC(OS16_No_EStops)XIC(G1_No_EStops)XIC(H1_No_EStops)OTE(LineSts.No_CTL_EStops);
   // --------------------------------------------System No Estops----------------------------------
   // Line Estop PB's OR System.No_Faults will cause the line to E-stop
   37: XIC(LineSts.No_CTC_EStops)XIC(LineSts.No_CTL_EStops)OTE(LineSts.No_Total_Estops);
   // -------Cut To Length Estop Timer---------------------------------------------------------------------------------
   // If an Estop is pressed the system will start counting down for X seconds, if the line is not at zero stop produce a coast stop.
   38: [XIO(LineSts.No_CTC_EStops) ,XIO(LineSts.No_CTC_Faults) ]TON(LineSts.CTCStopTimer,?,?);
   // ----------------------------------------Coast Stop Conditions----------------------------------------------------------
   // If the Estop Times out AND the line is not at Zero Speed then create a Coast Stop
   // If the Coast Stop PB is pressed then create a Coast
   39: [XIC(LineSts.CTCStopTimer.DN) ,XIC(Line_CTC_CoastStop) XIC(LineSts.ResetInput_CTC) XIO(Line_TotalMode) ]OTE(Line_CTC_CoastStop);
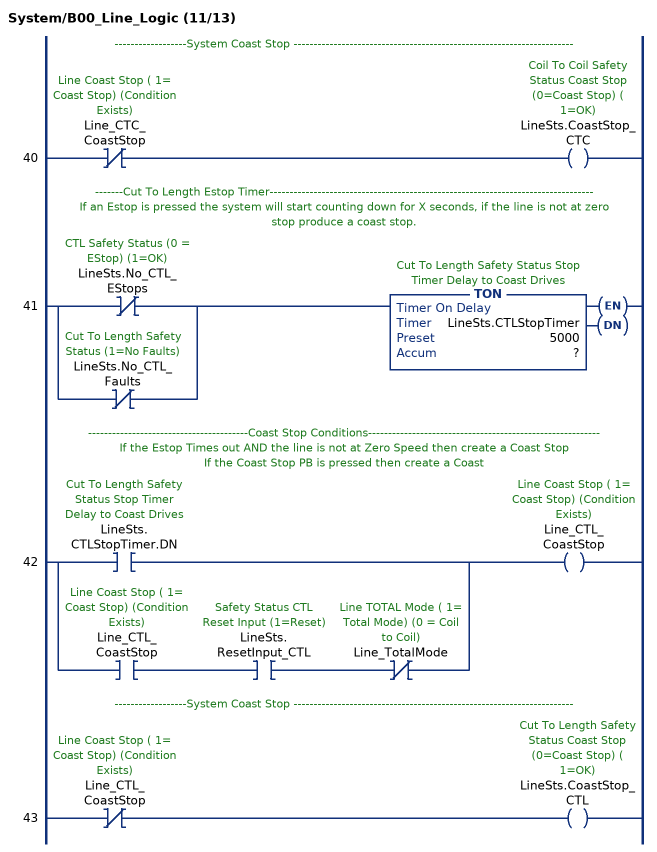
   // ------------------System Coast Stop ----------------------------------------------------------------------
   40: XIO(Line_CTC_CoastStop)OTE(LineSts.CoastStop_CTC);
   // -------Cut To Length Estop Timer---------------------------------------------------------------------------------
   // If an Estop is pressed the system will start counting down for X seconds, if the line is not at zero stop produce a coast stop.
   41: [XIO(LineSts.No_CTL_EStops) ,XIO(LineSts.No_CTL_Faults) ]TON(LineSts.CTLStopTimer,?,?);
   // ----------------------------------------Coast Stop Conditions----------------------------------------------------------
   // If the Estop Times out AND the line is not at Zero Speed then create a Coast Stop
   // If the Coast Stop PB is pressed then create a Coast
   42: [XIC(LineSts.CTLStopTimer.DN) ,XIC(Line_CTL_CoastStop) XIC(LineSts.ResetInput_CTL) XIO(Line_TotalMode) ]OTE(Line_CTL_CoastStop);
   // ------------------System Coast Stop ----------------------------------------------------------------------
   43: XIO(Line_CTL_CoastStop)OTE(LineSts.CoastStop_CTL);
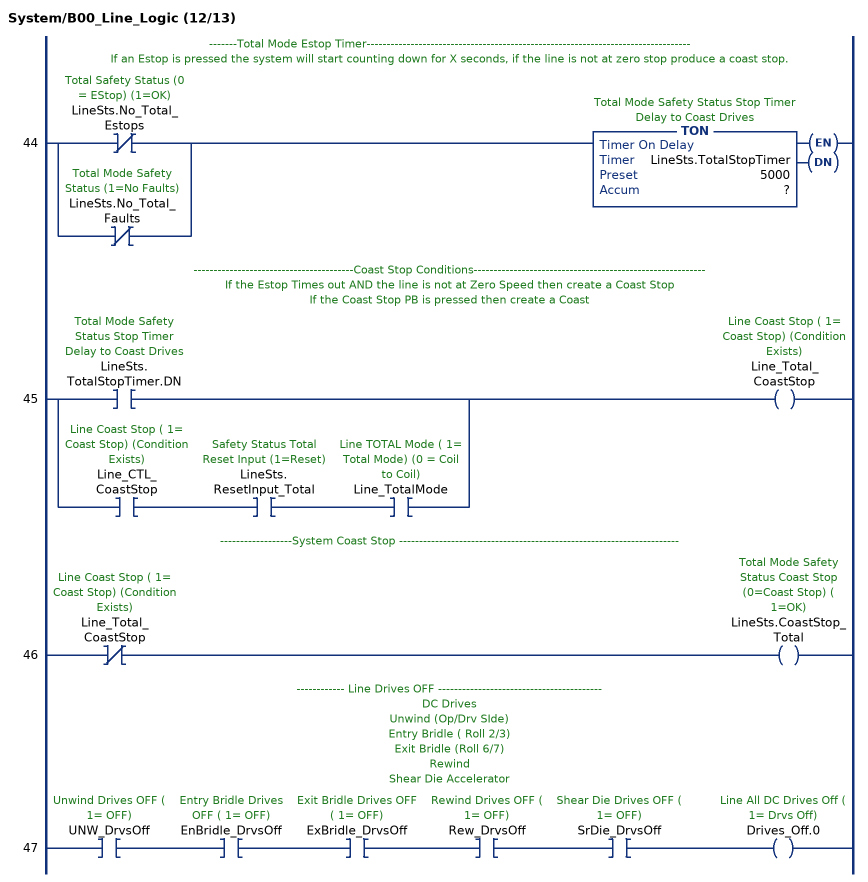
   // -------Total Mode Estop Timer---------------------------------------------------------------------------------
   // If an Estop is pressed the system will start counting down for X seconds, if the line is not at zero stop produce a coast stop.
   44: [XIO(LineSts.No_Total_Estops) ,XIO(LineSts.No_Total_Faults) ]TON(LineSts.TotalStopTimer,?,?);
   // ----------------------------------------Coast Stop Conditions----------------------------------------------------------
   // If the Estop Times out AND the line is not at Zero Speed then create a Coast Stop
   // If the Coast Stop PB is pressed then create a Coast
   45: [XIC(LineSts.TotalStopTimer.DN) ,XIC(Line_CTL_CoastStop) XIC(LineSts.ResetInput_Total) XIC(Line_TotalMode) ]OTE(Line_Total_CoastStop);
   // ------------------System Coast Stop ----------------------------------------------------------------------
   46: XIO(Line_Total_CoastStop)OTE(LineSts.CoastStop_Total);
   // ------------ Line Drives OFF -----------------------------------------
   // DC Drives
   // Unwind (Op/Drv SIde)
   // Entry Bridle ( Roll 2/3)
   // Exit Bridle (Roll 6/7)
   // Rewind
   // Shear Die Accelerator
   47: XIC(UNW_DrvsOff)XIC(EnBridle_DrvsOff)XIC(ExBridle_DrvsOff)XIC(Rew_DrvsOff)XIC(SrDie_DrvsOff)OTE(Drives_Off.0);
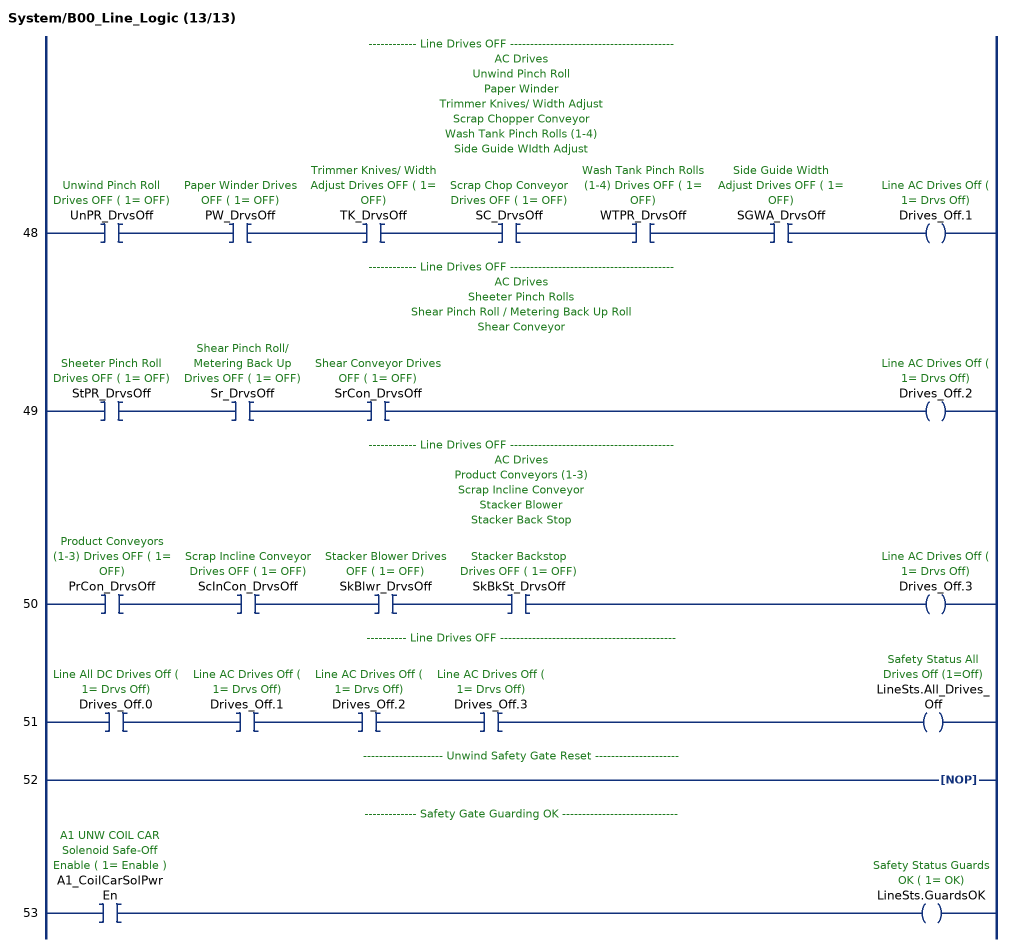
   // ------------ Line Drives OFF -----------------------------------------
   // AC Drives
   // Unwind Pinch Roll
   // Paper Winder
   // Trimmer Knives/ Width Adjust
   // Scrap Chopper Conveyor
   // Wash Tank Pinch Rolls (1-4)
   // Side Guide WIdth Adjust
   48: XIC(UnPR_DrvsOff)XIC(PW_DrvsOff)XIC(TK_DrvsOff)XIC(SC_DrvsOff)XIC(WTPR_DrvsOff)XIC(SGWA_DrvsOff)OTE(Drives_Off.1);
   // ------------ Line Drives OFF -----------------------------------------
   // AC Drives
   // Sheeter Pinch Rolls
   // Shear Pinch Roll / Metering Back Up Roll
   // Shear Conveyor
   49: XIC(StPR_DrvsOff)XIC(Sr_DrvsOff)XIC(SrCon_DrvsOff)OTE(Drives_Off.2);
   // ------------ Line Drives OFF -----------------------------------------
   // AC Drives
   // Product Conveyors (1-3)
   // Scrap Incline Conveyor
   // Stacker Blower
   // Stacker Back Stop
   50: XIC(PrCon_DrvsOff)XIC(ScInCon_DrvsOff)XIC(SkBlwr_DrvsOff)XIC(SkBkSt_DrvsOff)OTE(Drives_Off.3);
   // ---------- Line Drives OFF --------------------------------------------
   51: XIC(Drives_Off.0)XIC(Drives_Off.1)XIC(Drives_Off.2)XIC(Drives_Off.3)OTE(LineSts.All_Drives_Off);
   // -------------------- Unwind Safety Gate Reset ---------------------
   52: NOP();
   // ------------- Safety Gate Guarding OK -----------------------------
   53: XIC(A1_CoilCarSolPwrEn)OTE(LineSts.GuardsOK);
END_ROUTINE

ROUTINE C00_Shear_Logic   (* ladder *)
// Shear System
// Safety Logic
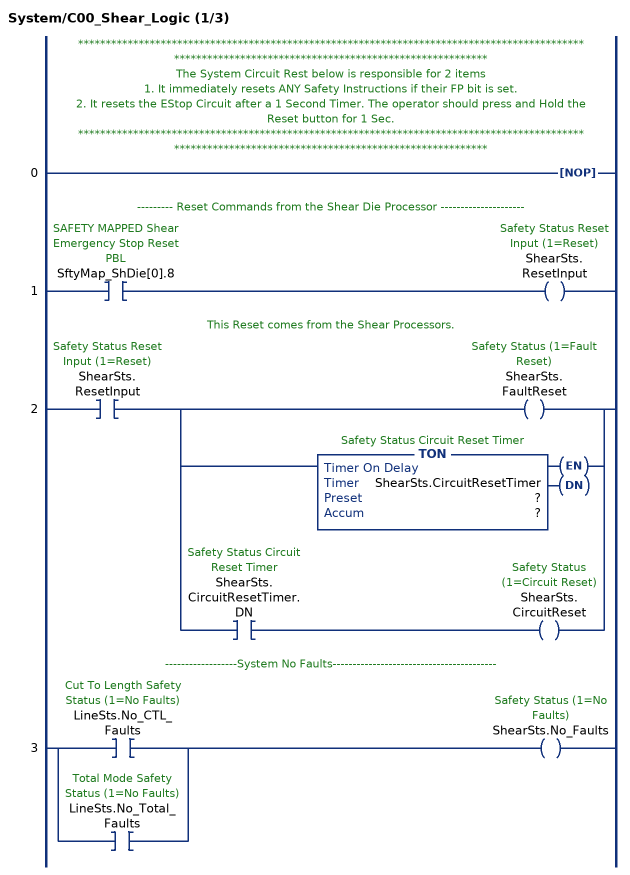
   // *****************************************************************************************************************************************************
   // The System Circuit Rest below is responsible for 2 items
   // 1. It immediately resets ANY Safety Instructions if their FP bit is set.
   // 2. It resets the EStop Circuit after a 1 Second Timer. The operator should press and Hold the Reset button for 1 Sec.
   // *****************************************************************************************************************************************************
   0: NOP();
   // --------- Reset Commands from the Shear Die Processor ---------------------
   1: XIC(SftyMap_ShDie[0].8)OTE(ShearSts.ResetInput);
   // This Reset comes from the Shear Processors.
   2: XIC(ShearSts.ResetInput)[OTE(ShearSts.FaultReset) ,TON(ShearSts.CircuitResetTimer,?,?) ,XIC(ShearSts.CircuitResetTimer.DN) OTE(ShearSts.CircuitReset) ];
   // ------------------System No Faults-----------------------------------------
   3: [XIC(LineSts.No_CTL_Faults) ,XIC(LineSts.No_Total_Faults) ]OTE(ShearSts.No_Faults);
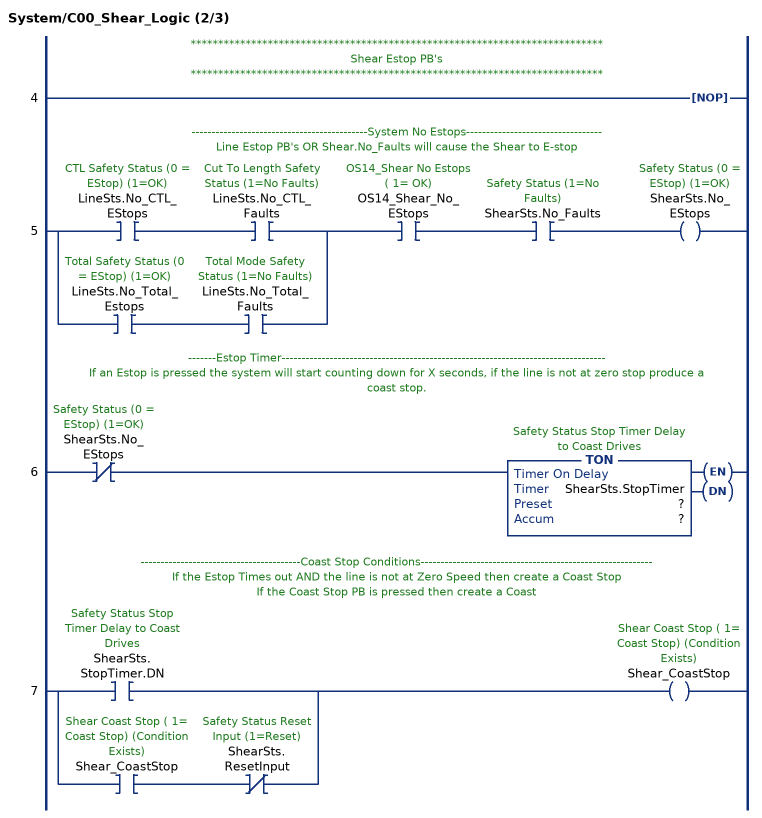
   // ***************************************************************************
   // Shear Estop PB's
   // ***************************************************************************
   4: NOP();
   // --------------------------------------------System No Estops----------------------------------
   // Line Estop PB's OR Shear.No_Faults will cause the Shear to E-stop
   5: [XIC(LineSts.No_CTL_EStops) XIC(LineSts.No_CTL_Faults) ,XIC(LineSts.No_Total_Estops) XIC(LineSts.No_Total_Faults) ]XIC(OS14_Shear_No_EStops)XIC(ShearSts.No_Faults)OTE(ShearSts.No_EStops);
   // -------Estop Timer---------------------------------------------------------------------------------
   // If an Estop is pressed the system will start counting down for X seconds, if the line is not at zero stop produce a coast stop.
   6: XIO(ShearSts.No_EStops)TON(ShearSts.StopTimer,?,?);
   // ----------------------------------------Coast Stop Conditions----------------------------------------------------------
   // If the Estop Times out AND the line is not at Zero Speed then create a Coast Stop
   // If the Coast Stop PB is pressed then create a Coast
   7: [XIC(ShearSts.StopTimer.DN) ,XIC(Shear_CoastStop) XIO(ShearSts.ResetInput) ]OTE(Shear_CoastStop);
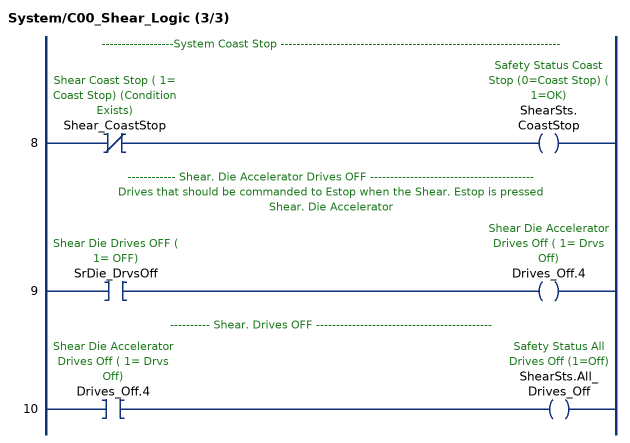
   // ------------------System Coast Stop ----------------------------------------------------------------------
   8: XIO(Shear_CoastStop)OTE(ShearSts.CoastStop);
   // ------------ Shear. Die Accelerator Drives OFF -----------------------------------------
   // Drives that should be commanded to Estop when the Shear. Estop is pressed
   // Shear. Die Accelerator
   9: XIC(SrDie_DrvsOff)OTE(Drives_Off.4);
   // ---------- Shear. Drives OFF --------------------------------------------
   10: XIC(Drives_Off.4)OTE(ShearSts.All_Drives_Off);
END_ROUTINE
